GLOBALCONSTANTS LED_FREQ (* Global constants *)
  (* Standard: 61499-1 *)
  (* Version 1.0, 2025-07-30, Franz Höpfinger *)
  PACKAGE logiBUS::io::DO_LED;
  VAR_GLOBAL CONSTANT
    LED_5HZ : UINT := 6; (* LED blinking 5HZ, highest Prio (Prio 6) *)
    LED_2HZ : UINT := 5; (* Identifier for LED blinking 2HZ, Prio 5 *)
    LED_1HZ : UINT := 4; (* Identifier for LED blinking 1HZ, Prio 4 *)
    LED_05HZ : UINT := 3; (* Identifier for LED blinking 0.5Hz, Prio 3 *)
    LED_breathing_05HZ : UINT := 2; (* Identifier for LED breathing 0.5HZ, Prio 2 *)
    LED_ON : UINT := 1; (* Identifier for LED always on, Prio 1 *)
    LED_OFF : UINT := 0; (* not used, reserved. *)
  END_VAR
END_GLOBALCONSTANTS
